FUNCTION_BLOCK 
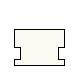
  EVENT_INPUT
    ;
  END_EVENT
  EVENT_OUTPUT
    ;
    ;
  END_EVENT
  VAR_INPUT
     : ;
     : ;
     : ;
     : ;
     : ;
  END_VAR
  VAR_OUTPUT
     : ;
     : ;
     : ;
     : ;
  END_VAR
  ALGORITHM ALG IN ST:

  END_ALGORITHM
END_FUNCTION_BLOCK
(* other elements stored in the file *)
(* ECState name=START Initial=true *)
(* ECState name=BODY *)
(* ECAction Algorithm=ALG *)
(* ECTransition Source=START Destination=BODY *)
(* ECEventCondition Event=EP3 *)
(* ECTransition Source=BODY Destination=EP4_STATE *)
(* ECCondition  (LS >= LS3) *)
(* ECState Name=EP4_STATE *)
(* ECAction Output=EP4 *)
(* ECTransition Source=BODY Destination=EP5_STATE *)
(* ECCondition  ((pH >= pHMin) AND (pH <= pHMax)) *)
(* ECState Name=EP5_STATE *)
(* ECAction Output=EP5 *)
